FUNCTION_BLOCK FB_LT_DT (* IEC 61131-3,Table 28#9 *)
  (* Standard: IEC 61499 *)
  (* Version 0.1, 2006-09-14, JHC, Holobloc Inc, Moved to fb.rt.compare. *)
  (* Version 0.0, 2004-12-15, JHC, Rockwell Automation, Converted from SRC format. *)
  (* Compiler header: package fb.rt.compare; *)
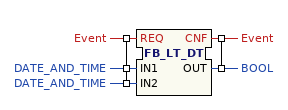
  EVENT_INPUT
    REQ WITH IN1, IN2;
  END_EVENT
  EVENT_OUTPUT
    CNF WITH OUT;
  END_EVENT
  VAR_INPUT
    IN1 : DATE_AND_TIME;
    IN2 : DATE_AND_TIME;
  END_VAR
  VAR_OUTPUT
    OUT : BOOL;
  END_VAR
END_FUNCTION_BLOCK
